PROGRAM A_Master
VAR

	// Buttons One-Shot Triggers:
	rtrigStartButton					:Tc2_Standard.R_TRIG;
	ftrigStartButton					:Tc2_Standard.F_TRIG;
	rtrigResetButton					:Tc2_Standard.R_TRIG;
	ftrigResetButton					:Tc2_Standard.F_TRIG;	
	rtrigStopButton					    :Tc2_Standard.R_TRIG;
	ftrigStopButton					    :Tc2_Standard.F_TRIG;

	
	//Write Persistent Data 
	fbWritePersistent					:Tc2_Utilities.FB_WritePersistentData;
	tonWritePeristentTrig				:Tc2_Standard.TON;
	bWritePersistentTrigger				:BOOL;	
	bWritePersistentError				:BOOL;
	bWritePersistentBusy				:BOOL;
	bWritePersistentErrID				:UDINT;
	tWritePersistentPeriod				:TIME := T#1M;	
	
	//----------------------------------------------------------------oldschoo1
	fbEventLogger						:	FB_EventLog;
	i                       :INT; //Int to handle user log index	
	k						:INT; //Int to handle user log index
	j						:INT;
	l						:INT;
	
END_VAR

// System PowerUP CTRL
tonSystemPowerUP(IN:=bSystemPoweringUP, PT:=tSystemPowerUP_Time);
IF tonSystemPowerUP.Q THEN 
bSystemPoweringUP:=FALSE;
 END_IF

tonFirstRun( IN := bFirstRun, PT := T#1S);

//
// Call Module's Actions:
			a_Map_Inputs();
	   b_Map_CtrlButtons();
	   
		  d_Call_Modules();
		  
		   f_Map_Outputs();
	   g_Map_StatusLamps();
  h_Write_PersistentData();
 			j_ManualMode();
  
//-------------------------oldschoo1

fbEventLogger(	bEnable       	:= PRG_MasterSystemTime.bReadyToRead AND NOT bSystemPoweringUP,
			    sDateTime     	:= PRG_MasterSystemTime.sDateTimeSpaces,
			    aEventFlags   	:= GVL_HMI.aEventFlags,
			    aEventTexts   	:= GVL_HMI.aEventTexts,
			    aActiveEvents 	:= GVL_HMI.aActiveEvents,
			    aEventLog     	:= GVL_HMI.aEventLog,
				siDate			:= GVL_MASTER.sSystemDate,
				siTime			:= GVL_MASTER.sSystemTime,
				soDate			:= GVL_HMI.aDateLog,
				soTime			:= GVL_HMI.aTimeLog
);

IF GVL_UTILITIES.bFlash250Hz THEN
FOR j := 0 TO 39 DO
	
GVL_HMI.stActiveEventsHMI[j].sActiveEvents := GVL_HMI.aActiveEvents[j];
END_FOR
FOR l:=0 TO 250 DO
	
	GVL_HMI.stAlarmHistory[l].sEventlog 	:= GVL_HMI.aEventLog[l];
	GVL_HMI.stAlarmHistory[l].sDate		:= GVL_HMI.aDateLog[l];
	GVL_HMI.stAlarmHistory[l].sTime		:= GVL_HMI.aTimeLog[l];
END_FOR
ELSE 
	
j:=0; 
l:=0;
END_IF

ACTION a_Map_Inputs:
// Safety Inputs
GVL_MASTER.stSafety.bSafety_OK						:= GVL_IO.isSafety_OK;
GVL_MASTER.stSafety.bDoorClosed						:= GVL_IO.isDoorClosed;
GVL_MASTER.stSafety.bDoorLocked						:= GVL_IO.isDoorLocked;
GVL_MASTER.stSafety.bEStop_OK						:= GVL_IO.isEStop_OK;
GVL_MASTER.stSafety.bLightBeam_Crossed				:= NOT GVL_IO.isLightBeam_NotCrossed;
GVL_MASTER.stSafety.bTwoHands_Signal				:= GVL_IO.isTwoHands_SIGNAL;



// Master Machine CTRL Inputs
GVL_MASTER.bPuck_Present							:= GVL_IO.iPuck_PresentSensor;
GVL_MASTER.bReservoir_Present						:= GVL_IO.iPartA_PresentSensor;
GVL_MASTER.bScrew_Present							:= GVL_IO.iPartB_PresentSensor;
GVL_MASTER.bGearBox_Present							:= GVL_IO.iPartC_PresentSensor;



// Y-Axis Inputs
GVL_MODULES.stY_Axis.bAxis_1_SafetyRelayFB			:= GVL_IO.iAxis_1_SafetyRelayFB;



// Kistler Inputs
GVL_MODULES.stKistler.st_TelegramDataIn				:= GVL_IO.iStatusBytes;
GVL_MODULES.stKistler.bKistlerCTRL_FB1				:= GVL_IO.iKistlerCTRL_FB1;						
GVL_MODULES.stKistler.bKistlerCTRL_FB2				:= GVL_IO.iKistlerCTRL_FB2;						 
GVL_MODULES.stKistler.bKistlerCTRL_FB3				:= GVL_IO.iKistlerCTRL_FB3;							



// Smac Inputs
GVL_MODULES.stSmac.bGripperA_ClosedSensor			:= GVL_IO.iGripperA_ClosedSensor;
GVL_MODULES.stSmac.bGripperB_ClosedSensor			:= GVL_IO.iGripperB_ClosedSensor;


//----------------------------------------------------------------------------------oldschoo1
END_ACTION

ACTION b_Map_CtrlButtons:

//Start button
rtrigStartButton(CLK:= GVL_IO.iStartButton,	Q=>bStartButtonRisingEdge);
ftrigStartButton(CLK:= GVL_IO.iStartButton,	Q=>bStartButtonFallingEdge);

// Stop button
rtrigStopButton(CLK:= NOT GVL_IO.iStopButton,  Q=>bStopButtonRisingEdge);
ftrigStopButton(CLK:= NOT GVL_IO.iStopButton,  Q=>bStopButtonFallingEdge);

// Reset button
rtrigResetButton(CLK:= GVL_IO.iResetButton, 	Q=>bResetButtonRisingEdge);
ftrigResetButton(CLK:= GVL_IO.iResetButton, 	Q=>bResetButtonFallingEdge);


//-------------------------------------------------------------------oldschoo1
END_ACTION

ACTION c_Read_Statuses:
//Handshake In
Y_Master_Y_Axis(STATUS => GVL_MODULES.Axis_STATUS);
K_Master_Kistler(STATUS => GVL_MODULES.Kistler_STATUS);
S_Master_SMAC(STATUS => GVL_MODULES.Smac_STATUS);
//--------------------------------------------oldschoo1
END_ACTION

ACTION d_Call_Modules:
// Call Modules Masters: ----------------------------------------*

			B_Safety();				// Safety PLC Module
							
	 c_Read_Statuses();
	  C_Machine_Ctrl();				// Master Module MachineCTRL
	 	e_Write_Cmds();
					
	 Y_Master_Y_Axis();				// Module for Y-Axis
   	   S_Master_SMAC();				// Module for Smac
	K_Master_Kistler();				// Module for Kistler	
   
//-------------------------------------------------------oldschoo1
END_ACTION

ACTION e_Write_Cmds:
//Handshake Out
Y_Master_Y_Axis(CMD := GVL_MODULES.CMD_Axis);
K_Master_Kistler(CMD := GVL_MODULES.CMD_Kistler);
S_Master_SMAC(CMD := GVL_MODULES.CMD_Smac);
//-----------------------------------------oldschoo1
END_ACTION

ACTION f_Map_Outputs:

// Safety Outputs
GVL_IO.qsSafetyRun								:= GVL_MASTER.stSafety.bRunSafety;
GVL_IO.qsSafetyErrorAck							:= GVL_MASTER.stSafety.bAckSafetyError;
GVL_IO.qsLockDoorCMD 							:= GVL_MASTER.stSafety.bLockDoor_CMD;
GVL_IO.qsLightBeam_MutingActive					:= GVL_MASTER.stSafety.bLightBeam_MuteCMD;
GVL_IO.qsTwoHandsMonitoring						:= GVL_MASTER.stSafety.bTwoHands_MonitorCMD;



// Master Machine CTRL Outputs
GVL_IO.qGripperA_Close							:= GVL_MODULES.stSmac.bGripperA_Close;
GVL_IO.qGripperA_Open							:= GVL_MODULES.stSmac.bGripperA_Open;
GVL_IO.qGripperB_Close							:= GVL_MODULES.stSmac.bGripperB_Close;
GVL_IO.qGripperB_Open							:= GVL_MODULES.stSmac.bGripperB_Open;
//GVL_IO.qCycleIndicator_GreenLED					:= GVL_MASTER.bCycleIndicator_Green;
//GVL_IO.qCycleIndicator_RedLED					:= GVL_MASTER.bCycleIndicator_Red;



// Y-Axis Outputs - 




// Kistler Outputs
GVL_IO.qControlBytes 							:= GVL_MODULES.stKistler.st_TelegramDataOut;
GVL_IO.qKistlerCTRL_Sig1						:= GVL_MODULES.stKistler.bKistlerCTRL_Sig1;
GVL_IO.qKistlerCTRL_Sig2						:= GVL_MODULES.stKistler.bKistlerCTRL_Sig2;
GVL_IO.qKistlerCTRL_Sig3						:= GVL_MODULES.stKistler.bKistlerCTRL_Sig3;
GVL_IO.qKistlerCTRL_Sig4						:= GVL_MODULES.stKistler.bKistlerCTRL_Sig4;



// Smac Outputs
GVL_IO.qGripperA_Open							:= GVL_MODULES.stSmac.bGripperA_Open;
GVL_IO.qGripperA_Close							:= GVL_MODULES.stSmac.bGripperA_Close;	
GVL_IO.qGripperB_Open							:= GVL_MODULES.stSmac.bGripperB_Open;
GVL_IO.qGripperB_Close							:= GVL_MODULES.stSmac.bGripperB_Close;

//---------------------------------------------------------------------------------------oldschoo1
END_ACTION

ACTION g_Map_StatusLamps:

// Reset Button LED Lamp
GVL_IO.qResetButton_LED := bFlash2Hz AND (stMachineStatus.bImmediateStopped OR 
								   		  stMachineStatus.bImmediateFault 	OR 
								          stMachineStatus.bCycleStopped 	OR
		   			 			          stMachineStatus.bCycleStopFault 	OR 
								          stMachineStatus.bInitialising);

		   
// Start Button LED Lamp
GVL_IO.qStartButton_LED := (stMachineStatus.bReadyToStart AND bFlash1Hz_7030) OR stMachineStatus.bAutoCycle;

(*
// Cycle Indicator LED Lamp
GVL_MASTER.bCycleIndicator_Green			:= stMachineStatus.bProcessCycle;
GVL_MASTER.bCycleIndicator_Red 				:= stMachineStatus.bAutoCycle AND NOT stMachineStatus.bProcessCycle; 
					
	*)
END_ACTION

ACTION h_Write_PersistentData:
tonWritePeristentTrig(IN := NOT bWritePersistentTrigger, 
					  PT := tWritePersistentPeriod, 
					  Q   => bWritePersistentTrigger);

fbWritePersistent(	NETID 	:= '', 
					PORT 	:= 851,
					START 	:= bWritePersistentTrigger,
					Mode 	:= E_PersistentMode.SPDM_2PASS,
					BUSY 	=> bWritePersistentBusy, 
					ERR 	=> bWritePersistentError,
					ERRID 	=> bWritePersistentErrID);
					
//----------------------------------------------------------oldschoo1
END_ACTION

ACTION i_TerminalInfo:

// TERMINAL 1 _ EK1100 - EtherCAT Coupler
GVL_IO.fbTerminalInfo[1](nTerminalState := GVL_IO.nEK1100State, 
sTerminalState => GVL_IO.sEK1100Status);
// TERMINAL 2 _ EL6070-0033	- License Key Terminal for TC3
GVL_IO.fbTerminalInfo[2](nTerminalState := GVL_IO.nEL6070State, 
sTerminalState => GVL_IO.sEL6070Status);
// TERMINAL 3 _ EL6910 - Safety PLC - Virtual Channels
GVL_IO.fbTerminalInfo[3](nTerminalState := GVL_IO.nEL6910State, 
sTerminalState => GVL_IO.sEL6910Status);
//TERMINAL 4 _ EL1918 - 8 Channel Digital Safety Inputs
GVL_IO.fbTerminalInfo[4](nTerminalState := GVL_IO.nEL1918_1State, 
sTerminalState => GVL_IO.sEL1918Status);
// TERMINAL 5 _ EL1918 - 8 Channel Digital Safety Inputs
GVL_IO.fbTerminalInfo[5](nTerminalState := GVL_IO.nEL1918_2State, 
sTerminalState => GVL_IO.sEL1918_2Status);
// TERMINAL 6 _ ELEL2904 - 4 Channel Digital Safety Outputs
GVL_IO.fbTerminalInfo[6](nTerminalState := GVL_IO.nEL2904_1State, 
sTerminalState => GVL_IO.sEL2904_1Status);
// TERMINAL 7 _ ELEL2904 - 4 Channel Digital Safety Outputs
GVL_IO.fbTerminalInfo[7](nTerminalState := GVL_IO.nEL2904_2State, 
sTerminalState => GVL_IO.sEL2904_2Status);
// TERMINAL 8 _ EL1809 - 16 Channel Digital Input Terminal
GVL_IO.fbTerminalInfo[8](nTerminalState := GVL_IO.nEL1809_1State, 
sTerminalState => GVL_IO.sEL1809_1Status);
// TERMINAL 9 _ EL1809 - 16 Channel Digital Input Terminal
GVL_IO.fbTerminalInfo[9](nTerminalState := GVL_IO.nEL1809_2State, 
sTerminalState => GVL_IO.sEL1809_2Status);
// TERMINAL 10 _ EL2809	- 16 Channel Digital Output Terminal
GVL_IO.fbTerminalInfo[10](nTerminalState := GVL_IO.nEL2809State, 
sTerminalState => GVL_IO.sEL2809Status);
// TERMINAL 11 _ EL9576 - Brake Chopper Terminal
GVL_IO.fbTerminalInfo[11](nTerminalState := GVL_IO.nEL9576State, 
sTerminalState => GVL_IO.sEL9576Status);
// TERMINAL 12 _ EL7211-0010 - Servo Motor Drive
GVL_IO.fbTerminalInfo[12](nTerminalState := GVL_IO.nEL7211State, 
sTerminalState => GVL_IO.sEL7211Status);
// BOX 13 _ maXYnos - Drive and Force Sensor for Kistler Press
GVL_IO.fbTerminalInfo[13](nTerminalState := GVL_IO.nKistlermaXYmosState, 
sTerminalState => GVL_IO.sKistlermaXYmosStatus);
END_ACTION

ACTION j_ManualMode:
IF	 GVL_MASTER.stMachineStatus.bReadyToStart THEN
	GVL_HMI.bEnableManualMode := TRUE;
ELSE GVL_HMI.bEnableManualMode := FALSE;
END_IF


GVL_HMI.rtrigManualMode(CLK:= GVL_HMI.nRegionMain=10 AND NOT GVL_HMI.rtrigManualModeOff[1].Q AND NOT GVL_HMI.rtrigManualModeOff[2].Q AND NOT GVL_HMI.rtrigManualModeOff[3].Q AND NOT GVL_HMI.rtrigManualModeOff[4].Q );
GVL_HMI.rtrigManualModeOff[1](CLK:=GVL_Master.stMachineStatus.bManualMode AND (GVL_HMI.nRegionMain <> 10));
GVL_HMI.rtrigManualModeOff[2](CLK:= rtrigStopButton.Q);
GVL_HMI.rtrigManualModeOff[3](CLK:= NOT GVL_Master.stMasterCTRL.bNoMachineImmediateFault );
GVL_HMI.rtrigManualModeOff[4](CLK := GVL_HMI.bManualModeOff[1], Q => GVL_HMI.bManualModeOff[2]);

IF GVL_HMI.rtrigManualMode.Q THEN 
	GVL_Master.stMasterCTRL.bManualModeRequest := TRUE;
	GVL_HMI.bManualModeOff[1] := FALSE;
ELSIF  GVL_HMI.rtrigManualModeOFF[1].Q OR  GVL_HMI.rtrigManualModeOFF[2].Q OR 
		GVL_HMI.rtrigManualModeOFF[3].Q THEN
		GVL_HMI.nRegionMain		:= 1;
	GVL_Master.stMasterCTRL.bManualModeRequest := FALSE ;
	GVL_HMI.bManualModeOff[1] := TRUE;
	
	
ELSE GVL_HMI.bManualModeOff[1] := FALSE;
	
END_IF
END_ACTION

END_PROGRAM

(* stored: Version 1.1.0.1, ProductVersion 3.1.4024.13
   POU A_Master: Id {bd8e4b1e-d504-48a9-bac3-34dbdf6704f4}, SpecialFunc None
   Action a_Map_Inputs: Id {197e0ebe-f91f-4144-bbed-a7377fbbe787}
   Action b_Map_CtrlButtons: Id {bb2c314f-2f9f-4b34-a2d7-bff4c9336f33}
   Action c_Read_Statuses: Id {82a8d1dd-2087-40e9-a1bf-2dcde5194972}
   Action d_Call_Modules: Id {d59654d5-a643-47f5-bf4b-9b6dbb2466da}
   Action e_Write_Cmds: Id {784f91b4-7272-4179-91fb-9a67e2781444}
   Action f_Map_Outputs: Id {80c55987-9b74-4f60-bc13-ffde7146848d}
   Action g_Map_StatusLamps: Id {360f6d9a-ca43-429e-82cb-bcaa758a6c8d}
   Action h_Write_PersistentData: Id {935fcb97-6522-48af-8ddf-ee1b01935492}
   Action i_TerminalInfo: Id {ad2881e6-f1aa-40c8-817f-9ef173460e64}
   Action j_ManualMode: Id {133cd35f-5fde-4a55-93c4-8067ca830846} *)
